// TIA Portal V19 export
FUNCTION_BLOCK "Rollformer_FB"   // FB183, LAD
TITLE = ROLLFORMER
// stored: MemoryReserve 100, SetENOAutomatically false
   VAR_INPUT
      AreaInterface : "AreaInterface";
      ZSI : "udt_ZoneSafetyInterface";
      DSI : "udt_DeviceSafetyInterface";
      Drive : "TAx_DriveInterface";
      DataIn : Struct
         Feed : "PositioningMachine_DataIn";
         ConnectorPlugged1 : Bool;
         ConnectorPlugged2 : Bool;
         ConnectorPlugged3Side1 : Bool;
         ConnectorPlugged3Side2 : Bool;
      END_STRUCT;
      CIn : Struct
         ExtEnable_LoopFwdOk : Bool;
         ExtEnable_LoopBwdOk : Bool;
         ExtEnable_FlyingShareOk : Bool;
         ExtEnable_MaterialCounterOK : Bool;
         ExtEnable_UnloadRollwayOk : Bool;
         ExtEnable_MwFakCalcOk : Bool;
         Loop1_VelOverride : LReal;
         SOS_Enable : Bool;
         Manager : "PositioningMachine_Manager";
      END_STRUCT;
      Config : Struct
         Feed : "PositioningMachine_Config";
         Data : "PositioningMachine_Ax_Parameters";
         DataPresence : Bool;
      END_STRUCT;
   END_VAR
   VAR_OUTPUT
      MachineInterface : "MachineInterface";
      COut : Struct
         Feed : "PositioningMachine_COut";
         EnableSOS : Bool;
      END_STRUCT;
      DataOut : Struct
         Feed : "PositioningMachine_DataOut";
      END_STRUCT;
   END_VAR
   VAR_IN_OUT
      TO_Ax : TO_PositioningAxis;
      PersistentValues : "udt_Rollformer_Pers";
   END_VAR
   VAR
      Alarms : Struct
         Feed : "PositioningMachine_Alr";
         ConnectorNotPlugged1 : Bool;
         ConnectorNotPlugged2 : Bool;
         ConnectorNotPlugged3Side1 : Bool;
         ConnectorNotPlugged3Side2 : Bool;
      END_STRUCT;
      Warnings : Struct
         Feed : "PositioningMachine_Wng";
         ExtraLowIsON : Bool;
         MissingCnd : Struct
            FlyingShare : Bool;
            MaterialCounter : Bool;
            UnloadRollway : Bool;
            MwFakClac : Bool;
            Loop1_Enable_BWD : Bool;
            Loop1_Enable_FWD : Bool;
         END_STRUCT;
      END_STRUCT;
      HMI : Struct
         MissingCnd : Struct
            FlyingShare : Bool;
            MaterialCounter : Bool;
            UnloadRollway : Bool;
            MwFacCalc : Bool;
            Loop1_Enable_BWD : Bool;
            Loop1_Enable_FWD : Bool;
         END_STRUCT;
         ManTargetMaterialPosition : LReal;
      END_STRUCT;
      Sts : Struct
         CndBWD_OK : Bool;
         CndFWD_OK : Bool;
      END_STRUCT;
      Feed : "PositioningMachine_FB";
      TON_SOS : TON_TIME;
   END_VAR
   VAR_TEMP
      Cnd : Bool;
      AdditionalWarnings : Bool;
      AdditionalAlarms : Bool;
      Req : Bool;
   END_VAR
   VAR CONSTANT
      AX_ENCODER_SMC30_MEAS_WHEEL : Int := 2;
   END_VAR
   VAR_TEMP   // added for the SCL form of the ladder/FBD networks
      _w1 : Bool;
      _w2 : Bool;
      _w3 : Bool;
      _w4 : Bool;
      _w5 : Bool;
      _w6 : Bool;
   END_VAR
BEGIN

REGION Network 1: >
END_REGION

REGION Network 2: Alarm wrong connector Plugged
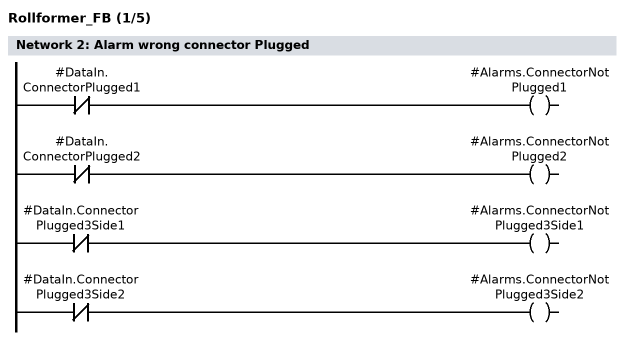
   RUNG wire#powerrail
      I_Contact( #DataIn.ConnectorPlugged1 )
      Coil( #Alarms.ConnectorNotPlugged1 )
   END_RUNG
   RUNG wire#powerrail
      I_Contact( #DataIn.ConnectorPlugged2 )
      Coil( #Alarms.ConnectorNotPlugged2 )
   END_RUNG
   RUNG wire#powerrail
      I_Contact( #DataIn.ConnectorPlugged3Side1 )
      Coil( #Alarms.ConnectorNotPlugged3Side1 )
   END_RUNG
   RUNG wire#powerrail
      I_Contact( #DataIn.ConnectorPlugged3Side2 )
      Coil( #Alarms.ConnectorNotPlugged3Side2 )
   END_RUNG
   // the same network as SCL:
   #Alarms.ConnectorNotPlugged1 := NOT #DataIn.ConnectorPlugged1;
   #Alarms.ConnectorNotPlugged2 := NOT #DataIn.ConnectorPlugged2;
   #Alarms.ConnectorNotPlugged3Side1 := NOT #DataIn.ConnectorPlugged3Side1;
   #Alarms.ConnectorNotPlugged3Side2 := NOT #DataIn.ConnectorPlugged3Side2;
END_REGION

REGION Network 3: Conditions HMI + Warnings + CIn
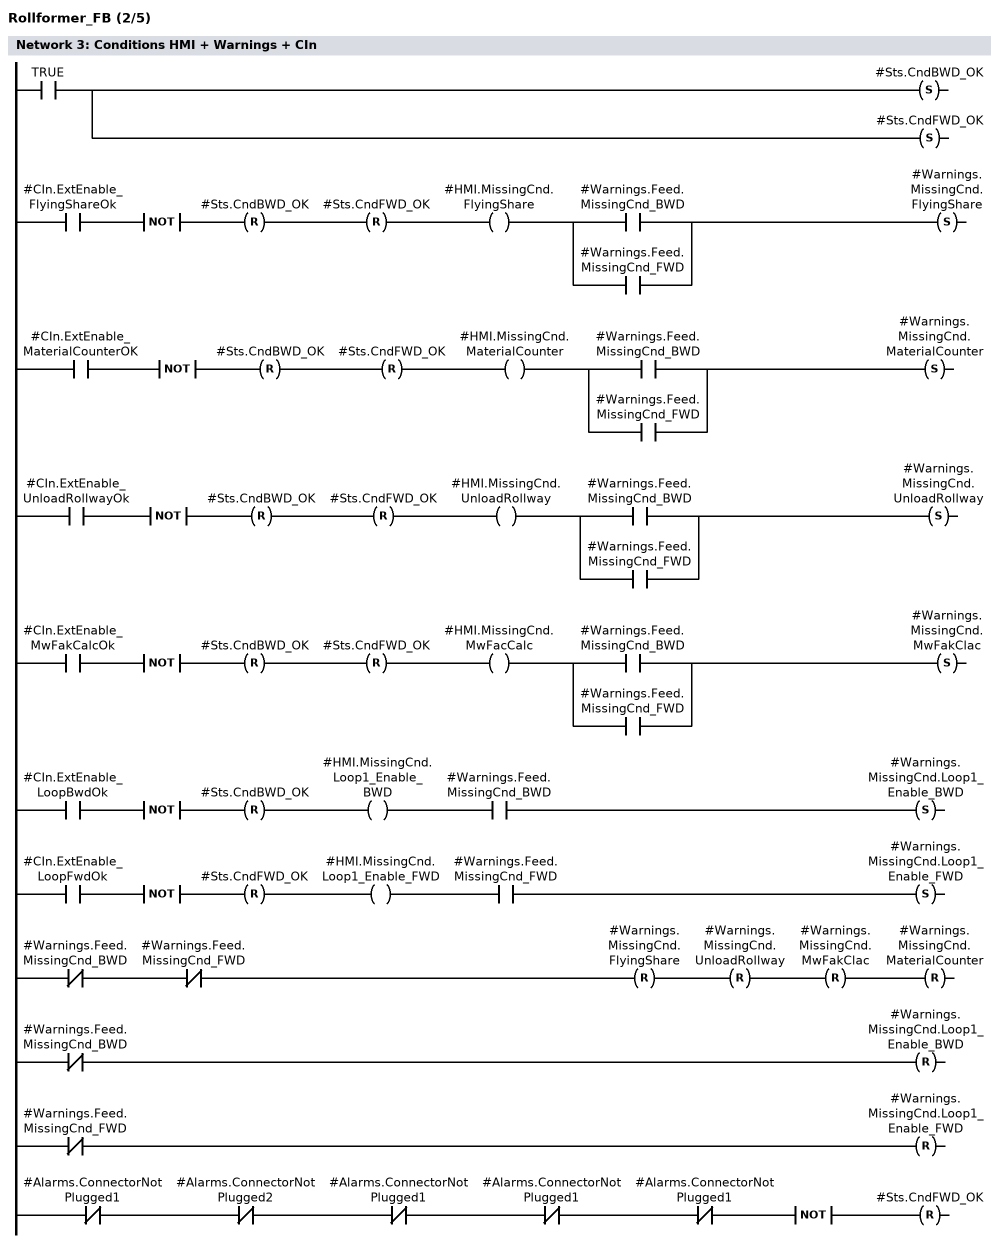
   RUNG wire#powerrail
      Contact( TRUE )
      wire#w1
      S_Coil( #Sts.CndBWD_OK )
   END_RUNG
   RUNG wire#w1
      S_Coil( #Sts.CndFWD_OK )
   END_RUNG
   RUNG wire#powerrail
      Contact( #CIn.ExtEnable_FlyingShareOk )
      Not()
      R_Coil( #Sts.CndBWD_OK )
      R_Coil( #Sts.CndFWD_OK )
      Coil( #HMI.MissingCnd.FlyingShare )
      wire#w2
      Contact( #Warnings.Feed.MissingCnd_BWD )
      wire#w3
      S_Coil( #Warnings.MissingCnd.FlyingShare )
   END_RUNG
   RUNG wire#w2
      Contact( #Warnings.Feed.MissingCnd_FWD )
   END_RUNG wire#w3
   RUNG wire#powerrail
      Contact( #CIn.ExtEnable_MaterialCounterOK )
      Not()
      R_Coil( #Sts.CndBWD_OK )
      R_Coil( #Sts.CndFWD_OK )
      Coil( #HMI.MissingCnd.MaterialCounter )
      wire#w4
      Contact( #Warnings.Feed.MissingCnd_BWD )
      wire#w5
      S_Coil( #Warnings.MissingCnd.MaterialCounter )
   END_RUNG
   RUNG wire#w4
      Contact( #Warnings.Feed.MissingCnd_FWD )
   END_RUNG wire#w5
   RUNG wire#powerrail
      Contact( #CIn.ExtEnable_UnloadRollwayOk )
      Not()
      R_Coil( #Sts.CndBWD_OK )
      R_Coil( #Sts.CndFWD_OK )
      Coil( #HMI.MissingCnd.UnloadRollway )
      wire#w6
      Contact( #Warnings.Feed.MissingCnd_BWD )
      wire#w7
      S_Coil( #Warnings.MissingCnd.UnloadRollway )
   END_RUNG
   RUNG wire#w6
      Contact( #Warnings.Feed.MissingCnd_FWD )
   END_RUNG wire#w7
   RUNG wire#powerrail
      Contact( #CIn.ExtEnable_MwFakCalcOk )
      Not()
      R_Coil( #Sts.CndBWD_OK )
      R_Coil( #Sts.CndFWD_OK )
      Coil( #HMI.MissingCnd.MwFacCalc )
      wire#w8
      Contact( #Warnings.Feed.MissingCnd_BWD )
      wire#w9
      S_Coil( #Warnings.MissingCnd.MwFakClac )
   END_RUNG
   RUNG wire#w8
      Contact( #Warnings.Feed.MissingCnd_FWD )
   END_RUNG wire#w9
   RUNG wire#powerrail
      Contact( #CIn.ExtEnable_LoopBwdOk )
      Not()
      R_Coil( #Sts.CndBWD_OK )
      Coil( #HMI.MissingCnd.Loop1_Enable_BWD )
      Contact( #Warnings.Feed.MissingCnd_BWD )
      S_Coil( #Warnings.MissingCnd.Loop1_Enable_BWD )
   END_RUNG
   RUNG wire#powerrail
      Contact( #CIn.ExtEnable_LoopFwdOk )
      Not()
      R_Coil( #Sts.CndFWD_OK )
      Coil( #HMI.MissingCnd.Loop1_Enable_FWD )
      Contact( #Warnings.Feed.MissingCnd_FWD )
      S_Coil( #Warnings.MissingCnd.Loop1_Enable_FWD )
   END_RUNG
   RUNG wire#powerrail
      I_Contact( #Warnings.Feed.MissingCnd_BWD )
      I_Contact( #Warnings.Feed.MissingCnd_FWD )
      R_Coil( #Warnings.MissingCnd.FlyingShare )
      R_Coil( #Warnings.MissingCnd.UnloadRollway )
      R_Coil( #Warnings.MissingCnd.MwFakClac )
      R_Coil( #Warnings.MissingCnd.MaterialCounter )
   END_RUNG
   RUNG wire#powerrail
      I_Contact( #Warnings.Feed.MissingCnd_BWD )
      R_Coil( #Warnings.MissingCnd.Loop1_Enable_BWD )
   END_RUNG
   RUNG wire#powerrail
      I_Contact( #Warnings.Feed.MissingCnd_FWD )
      R_Coil( #Warnings.MissingCnd.Loop1_Enable_FWD )
   END_RUNG
   RUNG wire#powerrail
      I_Contact( #Alarms.ConnectorNotPlugged1 )
      I_Contact( #Alarms.ConnectorNotPlugged2 )
      I_Contact( #Alarms.ConnectorNotPlugged1 )
      I_Contact( #Alarms.ConnectorNotPlugged1 )
      I_Contact( #Alarms.ConnectorNotPlugged1 )
      Not()
      R_Coil( #Sts.CndFWD_OK )
   END_RUNG
   // the same network as SCL:
   IF TRUE THEN
       #Sts.CndBWD_OK := TRUE;
       #Sts.CndFWD_OK := TRUE;
   END_IF;
   #_w1 := NOT #CIn.ExtEnable_FlyingShareOk;
   IF #_w1 THEN
       #Sts.CndBWD_OK := FALSE;
       #Sts.CndFWD_OK := FALSE;
   END_IF;
   #HMI.MissingCnd.FlyingShare := #_w1;
   IF #_w1 AND (#Warnings.Feed.MissingCnd_BWD OR #Warnings.Feed.MissingCnd_FWD) THEN
       #Warnings.MissingCnd.FlyingShare := TRUE;
   END_IF;
   #_w2 := NOT #CIn.ExtEnable_MaterialCounterOK;
   IF #_w2 THEN
       #Sts.CndBWD_OK := FALSE;
       #Sts.CndFWD_OK := FALSE;
   END_IF;
   #HMI.MissingCnd.MaterialCounter := #_w2;
   IF #_w2 AND (#Warnings.Feed.MissingCnd_BWD OR #Warnings.Feed.MissingCnd_FWD) THEN
       #Warnings.MissingCnd.MaterialCounter := TRUE;
   END_IF;
   #_w3 := NOT #CIn.ExtEnable_UnloadRollwayOk;
   IF #_w3 THEN
       #Sts.CndBWD_OK := FALSE;
       #Sts.CndFWD_OK := FALSE;
   END_IF;
   #HMI.MissingCnd.UnloadRollway := #_w3;
   IF #_w3 AND (#Warnings.Feed.MissingCnd_BWD OR #Warnings.Feed.MissingCnd_FWD) THEN
       #Warnings.MissingCnd.UnloadRollway := TRUE;
   END_IF;
   #_w4 := NOT #CIn.ExtEnable_MwFakCalcOk;
   IF #_w4 THEN
       #Sts.CndBWD_OK := FALSE;
       #Sts.CndFWD_OK := FALSE;
   END_IF;
   #HMI.MissingCnd.MwFacCalc := #_w4;
   IF #_w4 AND (#Warnings.Feed.MissingCnd_BWD OR #Warnings.Feed.MissingCnd_FWD) THEN
       #Warnings.MissingCnd.MwFakClac := TRUE;
   END_IF;
   #_w5 := NOT #CIn.ExtEnable_LoopBwdOk;
   IF #_w5 THEN #Sts.CndBWD_OK := FALSE; END_IF;
   #HMI.MissingCnd.Loop1_Enable_BWD := #_w5;
   IF #_w5 AND #Warnings.Feed.MissingCnd_BWD THEN #Warnings.MissingCnd.Loop1_Enable_BWD := TRUE; END_IF;
   #_w6 := NOT #CIn.ExtEnable_LoopFwdOk;
   IF #_w6 THEN #Sts.CndFWD_OK := FALSE; END_IF;
   #HMI.MissingCnd.Loop1_Enable_FWD := #_w6;
   IF #_w6 AND #Warnings.Feed.MissingCnd_FWD THEN #Warnings.MissingCnd.Loop1_Enable_FWD := TRUE; END_IF;
   IF NOT #Warnings.Feed.MissingCnd_BWD AND NOT #Warnings.Feed.MissingCnd_FWD THEN
       #Warnings.MissingCnd.FlyingShare := FALSE;
       #Warnings.MissingCnd.UnloadRollway := FALSE;
       #Warnings.MissingCnd.MwFakClac := FALSE;
       #Warnings.MissingCnd.MaterialCounter := FALSE;
   END_IF;
   IF NOT #Warnings.Feed.MissingCnd_BWD THEN #Warnings.MissingCnd.Loop1_Enable_BWD := FALSE; END_IF;
   IF NOT #Warnings.Feed.MissingCnd_FWD THEN #Warnings.MissingCnd.Loop1_Enable_FWD := FALSE; END_IF;
   IF NOT (NOT #Alarms.ConnectorNotPlugged1 AND NOT #Alarms.ConnectorNotPlugged2 AND NOT #Alarms.ConnectorNotPlugged1 AND NOT #Alarms.ConnectorNotPlugged1 AND NOT #Alarms.ConnectorNotPlugged1) THEN
       #Sts.CndFWD_OK := FALSE;
   END_IF;
END_REGION

REGION Network 4: COut - Enable SOS of S120 for avoiding material spring back while semiautomatic material threading
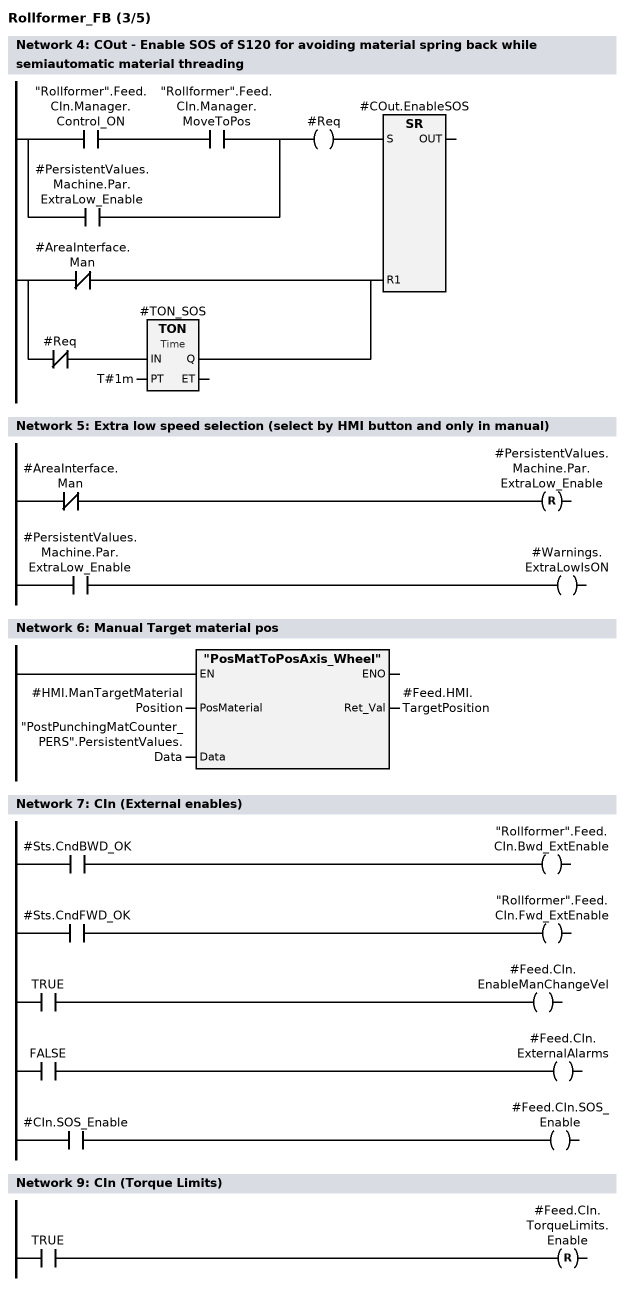
   RUNG wire#powerrail
      Contact( "Rollformer".Feed.CIn.Manager.Control_ON )
      Contact( "Rollformer".Feed.CIn.Manager.MoveToPos )
      wire#w1
      Coil( #Req )
      S_SR(operand := #COut.EnableSOS, r1 := wire#w2)
   END_RUNG
   RUNG wire#powerrail
      Contact( #PersistentValues.Machine.Par.ExtraLow_Enable )
   END_RUNG wire#w1
   RUNG wire#powerrail
      I_Contact( #AreaInterface.Man )
   END_RUNG wire#w2
   RUNG wire#powerrail
      I_Contact( #Req )
      { S7_Templates := "time_type := Time" } #TON_SOS.TON(pt := T#1m, et =>)
   END_RUNG wire#w2
   // the same network as SCL:
   #Req := ("Rollformer".Feed.CIn.Manager.Control_ON AND "Rollformer".Feed.CIn.Manager.MoveToPos) OR #PersistentValues.Machine.Par.ExtraLow_Enable;
   #TON_SOS(IN := NOT #Req, PT := T#1m);   // TON
   IF #Req THEN
       #COut.EnableSOS := TRUE;   // SR flip-flop
   END_IF;
   IF NOT #AreaInterface.Man OR #TON_SOS.Q THEN #COut.EnableSOS := FALSE; END_IF;
END_REGION

REGION Network 5: Extra low speed selection (select by HMI button and only in manual)
   RUNG wire#powerrail
      I_Contact( #AreaInterface.Man )
      R_Coil( #PersistentValues.Machine.Par.ExtraLow_Enable )
   END_RUNG
   RUNG wire#powerrail
      Contact( #PersistentValues.Machine.Par.ExtraLow_Enable )
      Coil( #Warnings.ExtraLowIsON )
   END_RUNG
   // the same network as SCL:
   IF NOT #AreaInterface.Man THEN #PersistentValues.Machine.Par.ExtraLow_Enable := FALSE; END_IF;
   #Warnings.ExtraLowIsON := #PersistentValues.Machine.Par.ExtraLow_Enable;
END_REGION

REGION Network 6: Manual Target material pos
   RUNG wire#powerrail
      "PosMatToPosAxis_Wheel"(PosMaterial := #HMI.ManTargetMaterialPosition, Data := "PostPunchingMatCounter_PERS".PersistentValues.Data, Ret_Val => #Feed.HMI.TargetPosition)
   END_RUNG
   // the same network as SCL:
   #Feed.HMI.TargetPosition := "PosMatToPosAxis_Wheel"(PosMaterial := #HMI.ManTargetMaterialPosition,
                           Data := "PostPunchingMatCounter_PERS".PersistentValues.Data);
END_REGION

REGION Network 7: CIn (External enables)
   RUNG wire#powerrail
      Contact( #Sts.CndBWD_OK )
      Coil( "Rollformer".Feed.CIn.Bwd_ExtEnable )
   END_RUNG
   RUNG wire#powerrail
      Contact( #Sts.CndFWD_OK )
      Coil( "Rollformer".Feed.CIn.Fwd_ExtEnable )
   END_RUNG
   RUNG wire#powerrail
      Contact( TRUE )
      Coil( #Feed.CIn.EnableManChangeVel )
   END_RUNG
   RUNG wire#powerrail
      Contact( FALSE )
      Coil( #Feed.CIn.ExternalAlarms )
   END_RUNG
   RUNG wire#powerrail
      Contact( #CIn.SOS_Enable )
      Coil( #Feed.CIn.SOS_Enable )
   END_RUNG
   // the same network as SCL:
   "Rollformer".Feed.CIn.Bwd_ExtEnable := #Sts.CndBWD_OK;
   "Rollformer".Feed.CIn.Fwd_ExtEnable := #Sts.CndFWD_OK;
   #Feed.CIn.EnableManChangeVel := TRUE;
   #Feed.CIn.ExternalAlarms := FALSE;
   #Feed.CIn.SOS_Enable := #CIn.SOS_Enable;
END_REGION

REGION Network 8 (SCL): CIn (Velocity override)
   #Feed.CIn.VelocityOverride.Enable := TRUE;
   #Feed.CIn.VelocityOverride.Value := 100.0;


   IF #PersistentValues.Machine.Par.ExtraLow_Enable AND #PersistentValues.Machine.Par.ExtraLow_VelPercentage > 0.0  THEN

       #Feed.CIn.VelocityOverride.Value := #PersistentValues.Machine.Par.ExtraLow_VelPercentage;

   END_IF;


   IF #AreaInterface.Cycle THEN

       IF #CIn.Loop1_VelOverride < #Feed.CIn.VelocityOverride.Value THEN
           #Feed.CIn.VelocityOverride.Value := #CIn.Loop1_VelOverride;
       END_IF;
   END_IF;
END_REGION

REGION Network 9: CIn (Torque Limits)
   RUNG wire#powerrail
      Contact( TRUE )
      R_Coil( #Feed.CIn.TorqueLimits.Enable )
   END_RUNG
   // the same network as SCL:
   IF TRUE THEN #Feed.CIn.TorqueLimits.Enable := FALSE; END_IF;
END_REGION

REGION Network 10: CIn (TO Parameters)
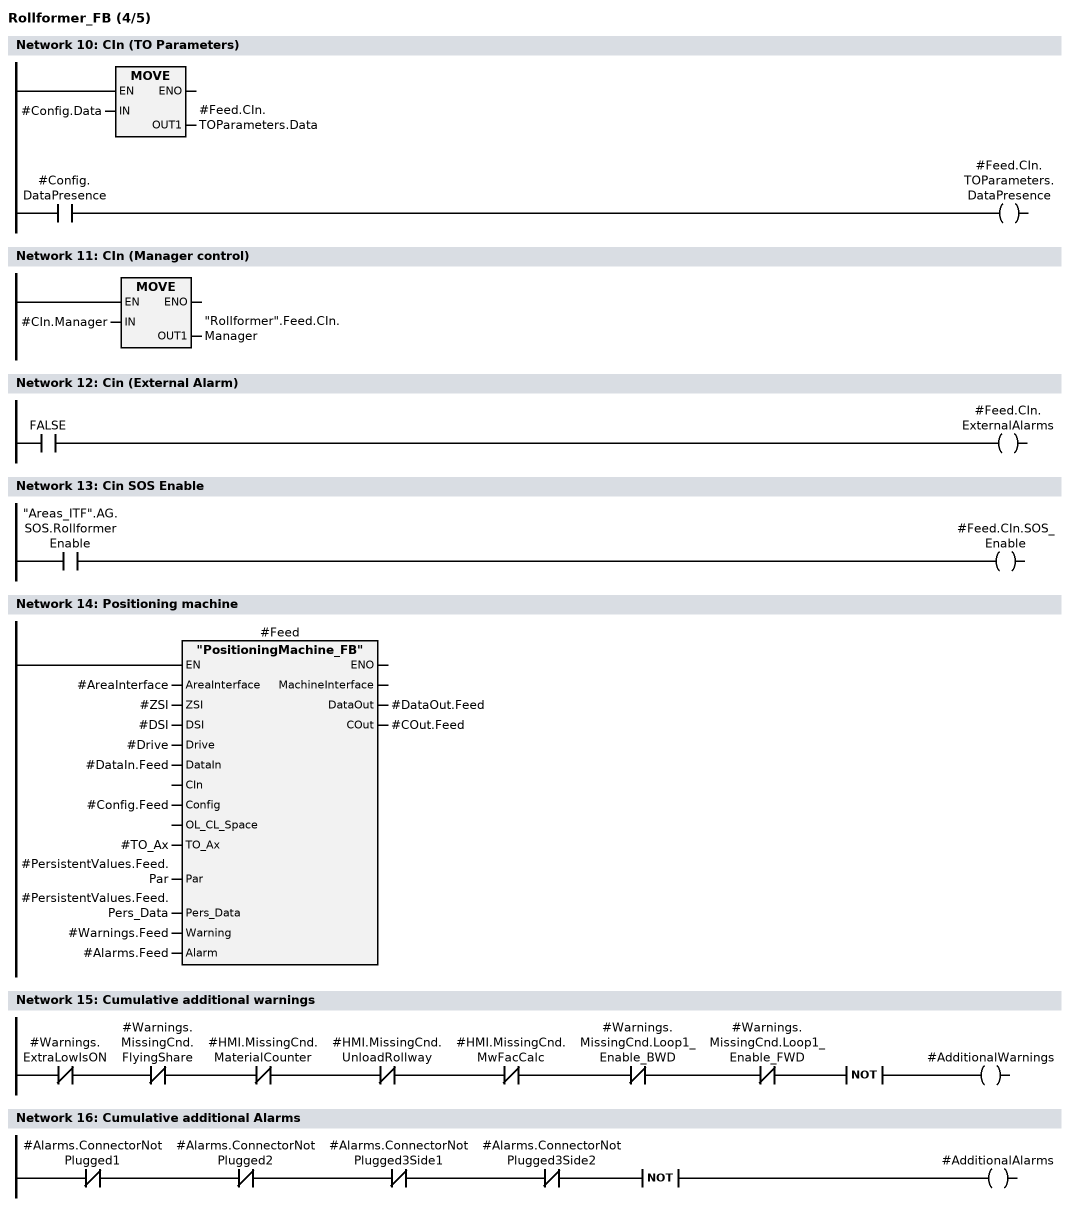
   RUNG wire#powerrail
      { S7_GenerateENO := "TRUE" } Move(in := #Config.Data, out1 => #Feed.CIn.TOParameters.Data)
   END_RUNG
   RUNG wire#powerrail
      Contact( #Config.DataPresence )
      Coil( #Feed.CIn.TOParameters.DataPresence )
   END_RUNG
   // the same network as SCL:
   #Feed.CIn.TOParameters.Data := #Config.Data;
   #Feed.CIn.TOParameters.DataPresence := #Config.DataPresence;
END_REGION

REGION Network 11: CIn (Manager control)
   RUNG wire#powerrail
      { S7_GenerateENO := "TRUE" } Move(in := #CIn.Manager, out1 => "Rollformer".Feed.CIn.Manager)
   END_RUNG
   // the same network as SCL:
   "Rollformer".Feed.CIn.Manager := #CIn.Manager;
END_REGION

REGION Network 12: Cin (External Alarm)
   RUNG wire#powerrail
      Contact( FALSE )
      Coil( #Feed.CIn.ExternalAlarms )
   END_RUNG
   // the same network as SCL:
   #Feed.CIn.ExternalAlarms := FALSE;
END_REGION

REGION Network 13: Cin SOS Enable
   RUNG wire#powerrail
      Contact( "Areas_ITF".AG.SOS.RollformerEnable )
      Coil( #Feed.CIn.SOS_Enable )
   END_RUNG
   // the same network as SCL:
   #Feed.CIn.SOS_Enable := "Areas_ITF".AG.SOS.RollformerEnable;
END_REGION

REGION Network 14: Positioning machine
   RUNG wire#powerrail
      #Feed(AreaInterface := #AreaInterface, ZSI := #ZSI, DSI := #DSI, Drive := #Drive, DataIn := #DataIn.Feed, CIn :=, Config := #Config.Feed, OL_CL_Space :=, TO_Ax := #TO_Ax, Par := #PersistentValues.Feed.Par, Pers_Data := #PersistentValues.Feed.Pers_Data, Warning := #Warnings.Feed, Alarm := #Alarms.Feed, MachineInterface =>, DataOut => #DataOut.Feed, COut => #COut.Feed)
   END_RUNG
   // the same network as SCL:
   #Feed(AreaInterface := #AreaInterface,   // "PositioningMachine_FB"
         ZSI := #ZSI,
         DSI := #DSI,
         Drive := #Drive,
         DataIn := #DataIn.Feed,
         Config := #Config.Feed,
         TO_Ax := #TO_Ax,
         Par := #PersistentValues.Feed.Par,
         Pers_Data := #PersistentValues.Feed.Pers_Data,
         Warning := #Warnings.Feed,
         Alarm := #Alarms.Feed,
         DataOut => #DataOut.Feed,
         COut => #COut.Feed);
END_REGION

REGION Network 15: Cumulative additional warnings
   RUNG wire#powerrail
      I_Contact( #Warnings.ExtraLowIsON )
      I_Contact( #Warnings.MissingCnd.FlyingShare )
      I_Contact( #HMI.MissingCnd.MaterialCounter )
      I_Contact( #HMI.MissingCnd.UnloadRollway )
      I_Contact( #HMI.MissingCnd.MwFacCalc )
      I_Contact( #Warnings.MissingCnd.Loop1_Enable_BWD )
      I_Contact( #Warnings.MissingCnd.Loop1_Enable_FWD )
      Not()
      Coil( #AdditionalWarnings )
   END_RUNG
   // the same network as SCL:
   #AdditionalWarnings := NOT (NOT #Warnings.ExtraLowIsON AND NOT #Warnings.MissingCnd.FlyingShare AND NOT #HMI.MissingCnd.MaterialCounter AND NOT #HMI.MissingCnd.UnloadRollway AND NOT #HMI.MissingCnd.MwFacCalc AND NOT #Warnings.MissingCnd.Loop1_Enable_BWD AND NOT #Warnings.MissingCnd.Loop1_Enable_FWD);
END_REGION

REGION Network 16: Cumulative additional Alarms
   RUNG wire#powerrail
      I_Contact( #Alarms.ConnectorNotPlugged1 )
      I_Contact( #Alarms.ConnectorNotPlugged2 )
      I_Contact( #Alarms.ConnectorNotPlugged3Side1 )
      I_Contact( #Alarms.ConnectorNotPlugged3Side2 )
      Not()
      Coil( #AdditionalAlarms )
   END_RUNG
   // the same network as SCL:
   #AdditionalAlarms := NOT (NOT #Alarms.ConnectorNotPlugged1 AND NOT #Alarms.ConnectorNotPlugged2 AND NOT #Alarms.ConnectorNotPlugged3Side1 AND NOT #Alarms.ConnectorNotPlugged3Side2);
END_REGION

REGION Network 17: >
END_REGION

REGION Network 18: >
END_REGION

REGION Network 19: Machine interface
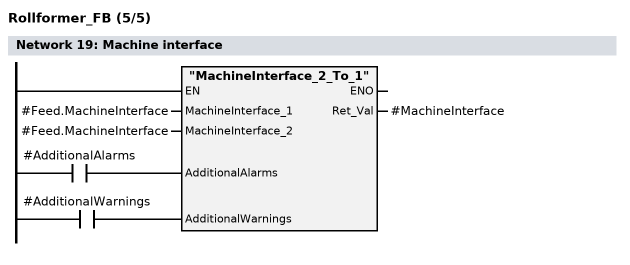
   RUNG wire#powerrail
      "MachineInterface_2_To_1"(AdditionalAlarms := wire#w1, AdditionalWarnings := wire#w2, MachineInterface_1 := #Feed.MachineInterface, MachineInterface_2 := #Feed.MachineInterface, Ret_Val => #MachineInterface)
   END_RUNG
   RUNG wire#powerrail
      Contact( #AdditionalAlarms )
   END_RUNG wire#w1
   RUNG wire#powerrail
      Contact( #AdditionalWarnings )
   END_RUNG wire#w2
   // the same network as SCL:
   #MachineInterface := "MachineInterface_2_To_1"(MachineInterface_1 := #Feed.MachineInterface,
                           MachineInterface_2 := #Feed.MachineInterface,
                           AdditionalAlarms := #AdditionalAlarms,
                           AdditionalWarnings := #AdditionalWarnings);
END_REGION

REGION Network 20: >
END_REGION

REGION Network 21: >
END_REGION
END_FUNCTION_BLOCK
